(* PLC project CHL-DZ-BJDX-11 宁波数字孪生（东方理工）研究院制备薄层色谱全自动化工作站_Old_InoProShop(V1.9.1.6).project, Inovance company InoProShop(V1.9.1.6) InoProShop(V1.9.1.6) *)
(* stored: creationDateTime 2026-06-16T17:55:18.1932567, modificationDateTime 2026-06-04T10:59:46 *)

VAR_GLOBAL  (* HMI_Date *)
  HMI_HandWheel_3Y : BOOL;  (* 手轮切换 *)
  HMI_HandWheel_4X : BOOL;
  HMI_HandWheel_5Z : BOOL;
  HMI_HandWheel_6X : BOOL;
  HMI_HandWheel_7Y : BOOL;
  HMI_HandWheel_8Y : BOOL;
  HMI_HandWheel_9X : BOOL;
  HMI_HandWheel_10Z : BOOL;
  HMI_HandWheel_11Y : BOOL;
  一键回原点 : BOOL;
  伺服上料_Setp : INT;
  伺服下料_Setp : INT;
  HMI_打样瓶上料轴3Y AT %MB132240 : HMI_Servo;  (* <GrpComment>\r\n <GrpComment_zh-cn><Sub/>{k:["[[1,10]]","position","write","execute"],s:{1:{t:"0",s:["1行","2行","3行","4行","5行","6行","上料位"]},2:{t:"0",s:["1行","2行","3行","4行","5行","6行","上料位"]},3:{t:"0",s:["1行","2行","3行","4行","5行","6行","上料位"]}}}</GrpComment_zh-cn>\r\n <GrpComment_1><Sub/></GrpComment_1>\r\n <GrpComment_2><Sub/></GrpComment_2>\r\n </GrpComment> *)
  HMI_点样轴6X AT %MB132344 : HMI_Servo;  (* <GrpComment>\r\n <GrpComment_zh-cn><Sub/>{k:["[[1,10]]","position","write","execute"],s:{1:{t:"0",s:["清洗位","起始位","终点位"]},2:{t:"0",s:["清洗位","起始位","终点位"]},3:{t:"0",s:["清洗位","起始位","终点位"]}}}</GrpComment_zh-cn>\r\n <GrpComment_1><Sub/></GrpComment_1>\r\n <GrpComment_2><Sub/></GrpComment_2>\r\n </GrpComment> *)
  HMI_点样轴7Y AT %MB132448 : HMI_Servo;  (* <GrpComment>\r\n <GrpComment_zh-cn><Sub/>{k:["[[1,10]]","position","write","execute"],s:{1:{t:"0",s:["放板位","起始位"]},2:{t:"0",s:["放板位","起始位"]},3:{t:"0",s:["放板位","起始位"]}}}</GrpComment_zh-cn>\r\n <GrpComment_1><Sub/></GrpComment_1>\r\n <GrpComment_2><Sub/></GrpComment_2>\r\n </GrpComment> *)
  HMI_地轨轴11Y AT %MB132552 : HMI_Servo;  (* <GrpComment>\r\n <GrpComment_zh-cn><Sub/>{k:["[[1,10]]","position","write","execute"],s:{1:{t:"0",s:["上样点样位","刮板拍照位","收集位","取工具位","展开位","取收集组位"]},2:{t:"0",s:["上样点样位","刮板拍照位","收集位","取工具位","展开位","取收集组位"]},3:{t:"0",s:["上样点样位","刮板拍照位","收集位","取工具位","展开位","取收集组位"]}}}\r\n </GrpComment_zh-cn>\r\n <GrpComment_1><Sub/></GrpComment_1>\r\n <GrpComment_2><Sub/></GrpComment_2>\r\n </GrpComment> *)
  HMI_上样轴4X轴 AT %MB132656 : HMI_Servo;  (* <GrpComment>\r\n <GrpComment_zh-cn><Sub/>{k:["[[1,10]]","position","write","execute"],s:{1:{t:"0",s:["1列","2列","3列","4列","5列","6列","7列","8列","清洗位"]},2:{t:"0",s:["1列","2列","3列","4列","5列","6列","7列","8列","清洗位"]},3:{t:"0",s:["1列","2列","3列","4列","5列","6列","7列","8列",\r\n "清洗位"]}}}</GrpComment_zh-cn>\r\n <GrpComment_1><Sub/></GrpComment_1>\r\n <GrpComment_2><Sub/></GrpComment_2>\r\n </GrpComment> *)
  HMI_上样轴5Z轴 AT %MB132760 : HMI_Servo;  (* <GrpComment>\r\n <GrpComment_zh-cn><Sub/>{k:["[[1,10]]","position","write","execute"],s:{1:{t:"0",s:["清洗位","上液位"]},2:{t:"0",s:["清洗位","上液位"]},3:{t:"0",s:["清洗位","上液位"]}}}</GrpComment_zh-cn>\r\n <GrpComment_1><Sub/></GrpComment_1>\r\n <GrpComment_2><Sub/></GrpComment_2>\r\n </GrpComment> *)
  收集流程 : INT;
  收集计数 : INT;
  展开流程 : INT;
  上样点样流程 : INT;
  拍照刮板流程 : INT;
  机器人流程 : INT;
  升降上料完成 AT %MB132040 : BOOL;
  升降下料完成 AT %MB132041 : BOOL;
  ECAT掉站报警 : BOOL;
END_VAR

VAR_GLOBAL  (* cyinder_date *)
  cyinderAlarm : INT;
  cyinderAlarm2 : INT;
  展缸1气缸1手动 : BOOL;
  展缸1气缸1自动 : BOOL;
  展缸1气缸2手动 : BOOL;
  展缸1气缸2自动 : BOOL;
  展缸1气缸3手动 : BOOL;
  展缸1气缸3自动 : BOOL;
  展缸1气缸4手动 : BOOL;
  展缸1气缸4自动 : BOOL;
  展缸2气缸1手动 : BOOL;
  展缸2气缸1自动 : BOOL;
  展缸2气缸2手动 : BOOL;
  展缸2气缸2自动 : BOOL;
  展缸2气缸3手动 : BOOL;
  展缸2气缸3自动 : BOOL;
  展缸2气缸4手动 : BOOL;
  展缸2气缸4自动 : BOOL;
  收集下压气缸手动 : BOOL;
  收集下压气缸自动 : BOOL;
  收集夹持气缸手动 : BOOL;
  收集夹持气缸自动 : BOOL;
  收集升降气缸手动 : BOOL;
  收集升降气缸自动 : BOOL;
  收集伸缩气缸手动 : BOOL;
  收集伸缩气缸自动 : BOOL;
  刮板拍照遮光气缸手动 : BOOL;
  刮板拍照遮光气缸自动 : BOOL;
  刮板拍照旋转气缸手动 : BOOL;
  刮板拍照旋转气缸自动 : BOOL;
  刮板拍照下压气缸手动 : BOOL;
  刮板拍照下压气缸自动 : BOOL;
  展缸1进液电池阀1手动 : BOOL;
  展缸1进液电池阀1自动 : BOOL;
  展缸1进液电池阀2手动 : BOOL;
  展缸1进液电池阀2自动 : BOOL;
  展缸1进液电池阀3手动 : BOOL;
  展缸1进液电池阀3自动 : BOOL;
  展缸1进液电池阀4手动 : BOOL;
  展缸1进液电池阀4自动 : BOOL;
  展缸1排液电池阀1手动 : BOOL;
  展缸1排液电池阀1自动 : BOOL;
  展缸1排液电池阀2手动 : BOOL;
  展缸1排液电池阀2自动 : BOOL;
  展缸1排液电池阀3手动 : BOOL;
  展缸1排液电池阀3自动 : BOOL;
  展缸1排液电池阀4手动 : BOOL;
  展缸1排液电池阀4自动 : BOOL;
  展缸1吹气电池阀1手动 : BOOL;
  展缸1吹气电池阀1自动 : BOOL;
  展缸1吹气电池阀2手动 : BOOL;
  展缸1吹气电池阀2自动 : BOOL;
  展缸1吹气电池阀3手动 : BOOL;
  展缸1吹气电池阀3自动 : BOOL;
  展缸1吹气电池阀4手动 : BOOL;
  展缸1吹气电池阀4自动 : BOOL;
  大真空泵手动 : BOOL;
  大真空泵自动 : BOOL;
  展缸2进液电池阀1手动 : BOOL;
  展缸2进液电池阀1自动 : BOOL;
  展缸2进液电池阀2手动 : BOOL;
  展缸2进液电池阀2自动 : BOOL;
  展缸2进液电池阀3手动 : BOOL;
  展缸2进液电池阀3自动 : BOOL;
  展缸2进液电池阀4手动 : BOOL;
  展缸2进液电池阀4自动 : BOOL;
  展缸2排液电池阀1手动 : BOOL;
  展缸2排液电池阀1自动 : BOOL;
  展缸2排液电池阀2手动 : BOOL;
  展缸2排液电池阀2自动 : BOOL;
  展缸2排液电池阀3手动 : BOOL;
  展缸2排液电池阀3自动 : BOOL;
  展缸2排液电池阀4手动 : BOOL;
  展缸2排液电池阀4自动 : BOOL;
  展缸2吹气电池阀1手动 : BOOL;
  展缸2吹气电池阀1自动 : BOOL;
  展缸2吹气电池阀2手动 : BOOL;
  展缸2吹气电池阀2自动 : BOOL;
  展缸2吹气电池阀3手动 : BOOL;
  展缸2吹气电池阀3自动 : BOOL;
  展缸2吹气电池阀4手动 : BOOL;
  展缸2吹气电池阀4自动 : BOOL;
  收集进液手动 : BOOL;
  收集进液自动 : BOOL;
  收集排液手动 : BOOL;
  收集排液自动 : BOOL;
  收集正压排液手动 : BOOL;
  收集正压排液自动 : BOOL;
  溶液收集瓶定位手动 : BOOL;
  溶液收集瓶定位自动 : BOOL;
  上样定位手动 : BOOL;
  上样定位自动 : BOOL;
  上样点样三通电池阀手动 : BOOL;
  上样点样三通电池阀自动 : BOOL;
  刮板拍照真空手动 : BOOL;
  刮板拍照真空自动 : BOOL;
  刮板拍照无刷电机手动 : BOOL;
  刮板拍照无刷电机自动 : BOOL;
  刮板拍照定位气缸手动 : BOOL;
  刮板拍照定位气缸自动 : BOOL;
  粉末收集器定位手动 : BOOL;
  粉末收集器定位自动 : BOOL;
  上样吹气手动 : BOOL;
  上样吹气自动 : BOOL;
END_VAR

VAR_GLOBAL  (* IO *)
  A相 AT %IX0.0 : BOOL;
  B相 AT %IX0.1 : BOOL;
  急停 AT %IX0.3 : BOOL;
  复位 AT %IX0.4 : BOOL;
  启动 AT %IX0.5 : BOOL;
  停止 AT %IX0.6 : BOOL;
  手自动 AT %IX0.7 : BOOL;
  倍率X1 AT %IX1.0 : BOOL;
  倍率X10 AT %IX1.1 : BOOL;
  倍率X100 AT %IX1.2 : BOOL;
  选择轴1 AT %IX1.3 : BOOL;
  选择轴2 AT %IX1.4 : BOOL;
  选择轴3 AT %IX1.5 : BOOL;
  选择轴4 AT %IX1.6 : BOOL;
  三色灯红 AT %QX0.0 : BOOL;
  三色灯黄 AT %QX0.1 : BOOL;
  三色灯绿 AT %QX0.2 : BOOL;
  蜂鸣器 AT %QX0.3 : BOOL;
  展缸1进液电池阀1 AT %QX1.0 : BOOL;
  展缸1进液电池阀2 AT %QX1.1 : BOOL;
  展缸1进液电池阀3 AT %QX1.2 : BOOL;
  展缸1进液电池阀4 AT %QX1.3 : BOOL;
  展缸1排液电池阀1 AT %QX1.4 : BOOL;
  展缸1排液电池阀2 AT %QX1.5 : BOOL;
  展缸1排液电池阀3 AT %QX1.6 : BOOL;
  展缸1排液电池阀4 AT %QX1.7 : BOOL;
  展缸1吹气电池阀1 AT %QX2.0 : BOOL;
  展缸1吹气电池阀2 AT %QX2.1 : BOOL;
  展缸1吹气电池阀3 AT %QX2.2 : BOOL;
  展缸1吹气电池阀4 AT %QX2.3 : BOOL;
  大真空泵 AT %QX2.4 : BOOL;
  展缸2进液电池阀1 AT %QX3.0 : BOOL;
  展缸2进液电池阀2 AT %QX3.1 : BOOL;
  展缸2进液电池阀3 AT %QX3.2 : BOOL;
  展缸2进液电池阀4 AT %QX3.3 : BOOL;
  展缸2排液电池阀1 AT %QX3.4 : BOOL;
  展缸2排液电池阀2 AT %QX3.5 : BOOL;
  展缸2排液电池阀3 AT %QX3.6 : BOOL;
  展缸2排液电池阀4 AT %QX3.7 : BOOL;
  展缸2吹气电池阀1 AT %QX4.0 : BOOL;
  展缸2吹气电池阀2 AT %QX4.1 : BOOL;
  展缸2吹气电池阀3 AT %QX4.2 : BOOL;
  展缸2吹气电池阀4 AT %QX4.3 : BOOL;
  收集平台进液2通电池阀 AT %QX5.0 : BOOL;
  收集平台排液3通电池阀 AT %QX5.1 : BOOL;
  收集平台正压排液阀 AT %QX5.2 : BOOL;
  溶液收集瓶工位定位气缸 AT %QX5.3 : BOOL;
  上样定位气缸 AT %QX7.0 : BOOL;
  上样点样三通电池阀 AT %QX7.1 : BOOL;
  刮板拍照真空阀 AT %QX7.2 : BOOL;
  刮板拍照无刷电机 AT %QX7.3 : BOOL;
  刮板拍照定位气缸 AT %QX7.4 : BOOL;
  粉末收集器工位定位气缸 AT %QX7.5 : BOOL;
  上样吹气二通阀 AT %QX7.6 : BOOL;
  展缸1气缸1原点 AT %IX3.0 : BOOL;
  展缸1气缸1动点 AT %IX3.1 : BOOL;
  展缸1气缸2原点 AT %IX3.2 : BOOL;
  展缸1气缸2动点 AT %IX3.3 : BOOL;
  展缸1气缸3原点 AT %IX3.4 : BOOL;
  展缸1气缸3动点 AT %IX3.5 : BOOL;
  展缸1气缸4原点 AT %IX3.6 : BOOL;
  展缸1气缸4动点 AT %IX3.7 : BOOL;
  展缸1排液气泡传感器 AT %IX4.0 : BOOL;
  展缸1溶剂废液检测传感器 AT %IX4.1 : BOOL;
  展缸2气缸1原点 AT %IX5.0 : BOOL;
  展缸2气缸1动点 AT %IX5.1 : BOOL;
  展缸2气缸2原点 AT %IX5.2 : BOOL;
  展缸2气缸2动点 AT %IX5.3 : BOOL;
  展缸2气缸3原点 AT %IX5.4 : BOOL;
  展缸2气缸3动点 AT %IX5.5 : BOOL;
  展缸2气缸4原点 AT %IX5.6 : BOOL;
  展缸2气缸4动点 AT %IX5.7 : BOOL;
  展缸2排液气泡传感器 AT %IX6.0 : BOOL;
  展缸2溶剂废液检测传感器 AT %IX6.1 : BOOL;
  收集平台下压气缸原点 AT %IX7.0 : BOOL;
  上料进料传感器 AT %IX7.1 : BOOL;
  收集平台夹持气缸原点 AT %IX7.2 : BOOL;
  收集平台夹持气缸动点 AT %IX7.3 : BOOL;
  收集平台升降气缸原点 AT %IX7.4 : BOOL;
  收集平台升降气缸动点 AT %IX7.5 : BOOL;
  收集平台推出气缸原点 AT %IX7.6 : BOOL;
  收集平台推出气缸动点 AT %IX7.7 : BOOL;
  收集平台气泡传感器 AT %IX8.0 : BOOL;
  收集平台瓶子有无传感器 AT %IX8.1 : BOOL;
  收集平台暂存工位传感器 AT %IX8.2 : BOOL;
  玻璃升降光电开关1 AT %IX8.3 : BOOL;
  玻璃升降光电开关2 AT %IX8.4 : BOOL;
  玻璃升降接近开关1 AT %IX8.5 : BOOL;
  玻璃升降接近开关2 AT %IX8.6 : BOOL;
  下料出料传感器 AT %IX8.7 : BOOL;
  上样料架检测1 AT %IX9.0 : BOOL;
  上样料架检测2 AT %IX9.1 : BOOL;
  上样气泡传感器 AT %IX9.2 : BOOL;
  点样气泡传感器 AT %IX9.3 : BOOL;
  刮板拍照遮光气缸上位 AT %IX9.4 : BOOL;
  刮板拍照遮光气缸下位 AT %IX9.5 : BOOL;
  刮板拍照旋转气缸原点 AT %IX9.6 : BOOL;
  刮板拍照旋转气缸动点 AT %IX9.7 : BOOL;
  刮板拍照下压气缸上位 AT %IX10.0 : BOOL;
  刮板拍照暂存工位传感器 AT %IX10.2 : BOOL;
  料库检测1 AT %IX11.0 : BOOL;
  料库检测2 AT %IX11.1 : BOOL;
  料库检测3 AT %IX11.2 : BOOL;
  料库检测4 AT %IX11.3 : BOOL;
  料库检测5 AT %IX11.4 : BOOL;
  料库检测6 AT %IX11.5 : BOOL;
  料库检测7 AT %IX11.6 : BOOL;
  料库检测8 AT %IX11.7 : BOOL;
  料库检测9 AT %IX12.0 : BOOL;
  料库检测10 AT %IX12.1 : BOOL;
  料库检测11 AT %IX12.2 : BOOL;
  料库检测12 AT %IX12.3 : BOOL;
  机器人工具检测1 AT %IX12.4 : BOOL;
  机器人工具检测2 AT %IX12.5 : BOOL;
  机器人工具检测3 AT %IX12.6 : BOOL;
END_VAR

VAR_GLOBAL RETAIN PERSISTENT  (* servoaxisdate *)
  玻璃上料轴1ZDATE AT %MB131072 : servo;
  玻璃上料轴2ZDATE AT %MB131160 : servo;
  打样瓶上料轴3YDATE AT %MB131248 : servo;
  点样轴6XDATE AT %MB131336 : servo;
  点样轴7YDATE AT %MB131424 : servo;
  拍照轴8YDATE AT %MB131512 : servo;
  刮板轴9XDATE AT %MB131600 : servo;
  刮板轴10ZDATE AT %MB131688 : servo;
  地轨轴11YDATE AT %MB131776 : servo;
  上样轴4X轴DATE AT %MB131864 : servo;
  上样轴5Z轴DATE AT %MB131952 : servo;
END_VAR

VAR_GLOBAL  (* GVL *)
  MODE_State : INT;
  Alarm : INT;  (* 0:停止 1:运行 2:故障 3:急停 *)
  ManualAuto : BOOL;
  初始化 : BOOL;
  转发转存 AT %MW1301 : STRING(128);
  接收字符 AT %MW1001 : STRING(128);
  CNC启动 : BOOL;
  CNC停止 : BOOL;
  CNC完成 : BOOL;
  伺服报警 : BOOL;
  回零完成1Z : BOOL;
  回零完成2Z : BOOL;
  回零完成3Y : BOOL;
  回零完成4X : BOOL;
  回零完成5Z : BOOL;
  回零完成6X : BOOL;
  回零完成7Y : BOOL;
  回零完成8Y : BOOL;
  回零完成9X : BOOL;
  回零完成10Z : BOOL;
  回零完成11Y : BOOL;
  伺服未回原点报警 : BOOL;
  collect_prepare_OK : BOOL;
  collect_OK : BOOL;
  Camera_scraper_initialization_OK : BOOL;
  Photo_preparation_completed_OK : BOOL;
  Scraper_collection_completed : BOOL;
  Robot_completes_material_retrieval : BOOL;
  Sampling_initialization_OK : BOOL;
  Sampling_Cleaning_OK : BOOL;
  Sampling_preparation_OK : BOOL;
  Sampling_Place_materials_OK : BOOL;
  Sampling_liquid_absorption : BOOL;
  Sampling_Spray_sample_OK : BOOL;
  expand_initialization_OK : BOOL;
  Expand_Group_clean_OK : BOOL;
  Expand_up_liquid_OK : BOOL;
  Expand_silica_gel_plate_OK : BOOL;
  排液开始 : BOOL;
  Collector_coordinates : INT;
  Collect_bottle_coordinates : INT;
  上样清洗位置 : INT;
  取工具setp : INT;
  取工具完成 : BOOL;
  取升降硅胶板step : INT;
  取升降硅胶板完成 : BOOL;
  放点样硅胶板step : INT;
  放点样硅胶板完成 : BOOL;
  取点样硅胶板step : INT;
  取点样硅胶板完成 : BOOL;
  放展缸硅胶板完成 : BOOL;
  放展缸硅胶板step : INT;
  取展缸硅胶板step : INT;
  取展缸硅胶板完成 : BOOL;
  放拍照硅胶板完成 : BOOL;
  放拍照硅胶板step : INT;
  取收集器组放暂存工位step : INT;
  取收集瓶组放暂存工位完成 : BOOL;
  取暂存收集器放刮板位完成 : BOOL;
  取暂存收集器放刮板位step : INT;
  取刮板收集器放到收集工位完成 : BOOL;
  取刮板收集器放到收集工位step : INT;
  取暂存收集瓶放收集工位step : INT;
  取暂存收集瓶放收集工位完成 : BOOL;
  取收集器放暂存工位完成 : BOOL;
  取收集器放暂存工位step : INT;
  取刮板硅胶板放废料区step : INT;
  取刮板硅胶板放废料区完成 : BOOL;
  取暂存收集器组放仓库完成 : BOOL;
  取暂存收集器组放仓库step : INT;
  取收集器组放暂存工位完成 : BOOL;
  取收集瓶组放暂存工位step : INT;
  取暂存收集瓶组放仓库完成 : BOOL;
  取暂存收集瓶组放仓库step : INT;
  取收集瓶放暂存工位step : INT;
  取收集瓶放暂存工位完成 : BOOL;
  B1 : ARRAY[1..2000] OF SMC_GEOINFO;
  泵站位符 : BOOL;
  B2 : ARRAY[1..2000] OF SMC_GEOINFO;
  DR : INT;
  大真空泵站位 : ARRAY[0..11] OF BOOL;
  取拍照硅胶完step : INT;
  取拍照硅胶板完成 : BOOL;
  上样料架报警 : BOOL;
  bParameterList1 : ARRAY[1..8] OF BOOL;
  Z1JOG_pos : BOOL;
  Z1JOG_neg : BOOL;
  Z2JOG_POS : BOOL;
  Z2JOG_NEG : BOOL;
END_VAR

VAR_GLOBAL  (* Host_Computer *)
  bOutput : BOOL;
  bEnable : BOOL := TRUE;
  bErrorReset : BOOL;
  bStepEnable : BOOL := TRUE;
  PLC_Busy : BOOL := FALSE;  (* <GrpComment>\r\n <GrpComment_zh-cn>PLC 正在执行动作</GrpComment_zh-cn>\r\n </GrpComment>\r\n PLC 正在执行动作 *)
  collect_Done : BOOL := FALSE;  (* <GrpComment>\r\n <GrpComment_zh-cn>修改:动作执行完成</GrpComment_zh-cn>\r\n </GrpComment>\r\n 修改:动作执行完成 *)
  collect_Error : BOOL := FALSE;  (* <GrpComment>\r\n <GrpComment_zh-cn>新增：动作执行错误/急停</GrpComment_zh-cn>\r\n </GrpComment>\r\n 新增：动作执行错误/急停 *)
  PLC_EStop : BOOL;  (* <GrpComment>\r\n <GrpComment_zh-cn>新增：急停</GrpComment_zh-cn>\r\n </GrpComment>\r\n 新增：急停 *)
  collect_Reset : BOOL;  (* <GrpComment>\r\n <GrpComment_zh-cn>新增：收集工位置位</GrpComment_zh-cn>\r\n </GrpComment>\r\n 新增：收集工位置位 *)
  collect_Step : INT;  (* <GrpComment>\r\n <GrpComment_zh-cn>修改：收集工位状态机</GrpComment_zh-cn>\r\n </GrpComment>\r\n 修改：收集工位状态机 *)
  collect_forward_instructions : STRING(128);  (* <GrpComment>\r\n <GrpComment_zh-cn>收集工位注射泵转发指令</GrpComment_zh-cn>\r\n </GrpComment>\r\n 收集工位注射泵转发指令 *)
  collect_count : INT;  (* <GrpComment>\r\n <GrpComment_zh-cn>收集次数</GrpComment_zh-cn>\r\n </GrpComment>\r\n 收集次数 *)
  collect_Enable : BOOL;  (* <GrpComment>\r\n <GrpComment_zh-cn>新增：收集工位启动</GrpComment_zh-cn>\r\n </GrpComment>\r\n 新增：收集工位启动 *)
  collect_Busy : BOOL;  (* <GrpComment>\r\n <GrpComment_zh-cn>新增：收集工位忙</GrpComment_zh-cn>\r\n </GrpComment>\r\n 新增：收集工位忙 *)
  Expand_Enable : BOOL;  (* <GrpComment>\r\n <GrpComment_zh-cn>PC→PLC: TRUE 启动状态机</GrpComment_zh-cn>\r\n </GrpComment>\r\n PC→PLC: TRUE 启动状态机 *)
  Expand_Step : INT;  (* <GrpComment>\r\n <GrpComment_zh-cn>PLC→PC: 子步号 {0,10,20,30,40,90}</GrpComment_zh-cn>\r\n </GrpComment>\r\n PLC→PC: 子步号 {0,10,20,30,40,90} *)
  Expand_Done : BOOL;  (* <GrpComment>\r\n <GrpComment_zh-cn>PLC→PC: prep完成锁存（语义变更：prep完成非整流程完成）</GrpComment_zh-cn>\r\n </GrpComment>\r\n PLC→PC: prep完成锁存（语义变更：prep完成非整流程完成） *)
  Expand_Error : BOOL;  (* <GrpComment>\r\n <GrpComment_zh-cn>PLC→PC: 故障锁存（Step=90），Expand_Reset=TRUE 清零</GrpComment_zh-cn>\r\n </GrpComment>\r\n PLC→PC: 故障锁存（Step=90），Expand_Reset=TRUE 清零 *)
  Expand_Reset : BOOL;  (* <GrpComment>\r\n <GrpComment_zh-cn>PC→PLC: TRUE 清错误</GrpComment_zh-cn>\r\n </GrpComment>\r\n PC→PLC: TRUE 清错误 *)
  Expand_Busy : BOOL;  (* <GrpComment>\r\n <GrpComment_zh-cn>PLC→PC: 派生 (Step∈[10,80]) AND NOT Done</GrpComment_zh-cn>\r\n </GrpComment>\r\n PLC→PC: 派生 (Step∈[10,80]) AND NOT Done *)
  Expand_Mode_Flag : INT;  (* <GrpComment>\r\n <GrpComment_zh-cn>0=缸模式润洗 / 1=管路模式润洗</GrpComment_zh-cn>\r\n </GrpComment>\r\n 0=缸模式润洗 / 1=管路模式润洗 *)
  Expand_Group : INT;  (* <GrpComment>\r\n <GrpComment_zh-cn>展开组号 (1 或 2)，由 PLC 自动推导</GrpComment_zh-cn>\r\n </GrpComment>\r\n 展开组号 (1 或 2)，由 PLC 自动推导 *)
  Expand_Number : INT;  (* <GrpComment>\r\n <GrpComment_zh-cn>缸号在组内序号（1-4），由 PLC 自动推导</GrpComment_zh-cn>\r\n </GrpComment>\r\n 缸号在组内序号（1-4），由 PLC 自动推导 *)
  Expand_up_liquid_count : INT;  (* <GrpComment>\r\n <GrpComment_zh-cn>注射泵 DT 协议指令（合并后的单一变量）</GrpComment_zh-cn>\r\n </GrpComment>\r\n 上液注射泵重复次数 *)
  Expand_rinse_count : INT;  (* <GrpComment>\r\n <GrpComment_zh-cn>注射泵 DT 协议指令（合并后的单一变量）</GrpComment_zh-cn>\r\n </GrpComment>\r\n 润洗重复次数 *)
  Expand_forward_instructions : STRING(128);  (* <GrpComment>\r\n <GrpComment_zh-cn>注射泵 DT 协议指令（合并后的单一变量）</GrpComment_zh-cn>\r\n </GrpComment>\r\n 注射泵 DT 协议指令（合并后的单一变量） *)
  Tank_State : ARRAY[1..8] OF INT;  (* <GrpComment>\r\n <GrpComment_zh-cn>══════════════════════════════════════════════════════════════\r\n 【新增】展缸状态跟踪\r\n ══════════════════════════════════════════════════════════════</GrpComment_zh-cn>\r\n </GrpComment>\r\n ══════════════════════════════════════════════════════════════\r\n 【新增】展缸状态跟踪\r\n ══════════════════════════════════════════════════════════════ *)
  Tank_SampleID : ARRAY[1..8] OF DINT;  (* <GrpComment>\r\n <GrpComment_zh-cn>PLC→PC: 每缸状态\r\n 0 = Idle（空闲，可分配）\r\n 10 = Prepping（准备中：润洗/上液/放板）\r\n 40 = Developing（展开中，等待视觉/延时触发排液）\r\n 50 = Draining（排液中）\r\n 99 = Done（排液完成，等待 PC 释放）\r\n 90 = Error（故障）</GrpComment_zh-cn>\r\n </GrpComment>\r\n PLC→PC: 每缸状态\r\n 0 = Idle（空闲，可分配）\r\n 10 = Prepping（准备中：润洗/上液/放板）\r\n 40 = Developing（展开中，等待视觉/延时触发排液）\r\n 50 = Draining（排液中）\r\n 99 = Done（排液完成，等待 PC 释放）\r\n 90 = Error（故障） *)
  Expand_Target_Tank : INT;  (* <GrpComment>\r\n <GrpComment_zh-cn>PC→PLC: 绑定样品 ID（调试/溯源用，PLC 不使用此值做逻辑判断）\r\n ══════════════════════════════════════════════════════════════\r\n 【新增】Prep 目标参数\r\n ══════════════════════════════════════════════════════════════</GrpComment_zh-cn>\r\n </GrpComment>\r\n PC→PLC: 绑定样品 ID（调试/溯源用，PLC 不使用此值做逻辑判断）\r\n ══════════════════════════════════════════════════════════════\r\n 【新增】Prep 目标参数\r\n ══════════════════════════════════════════════════════════════ *)
  Tank_Drain_Enable : ARRAY[1..8] OF BOOL;  (* <GrpComment>\r\n <GrpComment_zh-cn>PC→PLC: 目标缸号(1-8)，Enable 触发前写入\r\n PLC 读取后自动推导：\r\n Expand_Group = (Target_Tank - 1) / 4 + 1\r\n Expand_Number = (Target_Tank - 1) MOD 4 + 1\r\n ══════════════════════════════════════════════════════════════\r\n 【新增】Per-tank 排液控制\r\n ══════════════════════════════════════════════════════════════</GrpComment_zh-cn>\r\n </GrpComment>\r\n PC→PLC: 目标缸号(1-8)，Enable 触发前写入\r\n PLC 读取后自动推导：\r\n Expand_Group = (Target_Tank - 1) / 4 + 1\r\n Expand_Number = (Target_Tank - 1) MOD 4 + 1\r\n ══════════════════════════════════════════════════════════════\r\n 【新增】Per-tank 排液控制\r\n ══════════════════════════════════════════════════════════════ *)
  Tank_Drain_Done : ARRAY[1..8] OF BOOL;  (* <GrpComment>\r\n <GrpComment_zh-cn>PC→PLC: 触发第 i 缸排液（前置条件：Tank_State[i]=40）</GrpComment_zh-cn>\r\n </GrpComment>\r\n PC→PLC: 触发第 i 缸排液（前置条件：Tank_State[i]=40） *)
  DrainTimer : ARRAY[1..8] OF TON;  (* <GrpComment>\r\n <GrpComment_zh-cn>PLC→PC: 第 i 缸排液完成锁存\r\n PC 确认后写 Tank_Drain_Enable[i]=FALSE 进行复位\r\n ══════════════════════════════════════════════════════════════\r\n 【新增】排液子程序内部变量\r\n ══════════════════════════════════════════════════════════════</GrpComment_zh-cn>\r\n </GrpComment>\r\n PLC→PC: 第 i 缸排液完成锁存\r\n PC 确认后写 Tank_Drain_Enable[i]=FALSE 进行复位\r\n ══════════════════════════════════════════════════════════════\r\n 【新增】排液子程序内部变量\r\n ══════════════════════════════════════════════════════════════ *)
  DrainDuration : TIME := TIME#5s0ms;  (* <GrpComment>\r\n <GrpComment_zh-cn>每缸排液定时器（后续可替换为传感器判断）</GrpComment_zh-cn>\r\n </GrpComment>\r\n 每缸排液定时器（后续可替换为传感器判断） *)
  Sampling_Enable : BOOL;  (* <GrpComment>\r\n <GrpComment_zh-cn>PC→PLC: TRUE 启动状态机</GrpComment_zh-cn>\r\n </GrpComment>\r\n PC→PLC: TRUE 启动状态机 *)
  Sampling_Step : INT;  (* <GrpComment>\r\n <GrpComment_zh-cn>PLC→PC: 子步号 {0,10,20,30,40,50,90}</GrpComment_zh-cn>\r\n </GrpComment>\r\n PLC→PC: 子步号 {0,10,20,30,40,50,90} *)
  Sampling_Done : BOOL;  (* <GrpComment>\r\n <GrpComment_zh-cn>PLC→PC: 完成锁存（Step 50 结束后置 TRUE）</GrpComment_zh-cn>\r\n </GrpComment>\r\n PLC→PC: 完成锁存（Step 50 结束后置 TRUE） *)
  Sampling_Error : BOOL;  (* <GrpComment>\r\n <GrpComment_zh-cn>PLC→PC: 故障锁存（Step=90），Sampling_Reset=TRUE 清零</GrpComment_zh-cn>\r\n </GrpComment>\r\n PLC→PC: 故障锁存（Step=90），Sampling_Reset=TRUE 清零 *)
  Sampling_Reset : BOOL;  (* <GrpComment>\r\n <GrpComment_zh-cn>PC→PLC: TRUE 清错误</GrpComment_zh-cn>\r\n </GrpComment>\r\n PC→PLC: TRUE 清错误 *)
  Sampling_Busy : BOOL;  (* <GrpComment>\r\n <GrpComment_zh-cn>PLC→PC: 派生 (Step∈[10,80]) AND NOT Done</GrpComment_zh-cn>\r\n </GrpComment>\r\n PLC→PC: 派生 (Step∈[10,80]) AND NOT Done *)
  Sampling_clean_instructions : ARRAY[1..2] OF STRING(128);  (* <GrpComment>\r\n <GrpComment_zh-cn>PC→PLC: 清洗泵指令（1条DT协议）</GrpComment_zh-cn>\r\n </GrpComment>\r\n PC→PLC: 清洗泵指令（1条DT协议） *)
  Sampling_clean_count : INT;  (* <GrpComment>\r\n <GrpComment_zh-cn>PC→PLC: 清洗次数（0=跳过清洗）</GrpComment_zh-cn>\r\n </GrpComment>\r\n PC→PLC: 清洗次数（0=跳过清洗） *)
  Sampling_prep_instructions : ARRAY[1..2] OF STRING(128);  (* <GrpComment>\r\n <GrpComment_zh-cn>── Step 20 气泡准备 ──</GrpComment_zh-cn>\r\n </GrpComment>\r\n 上样准备泵指令 *)
  Sampling_bubble_count : INT;  (* <GrpComment>\r\n <GrpComment_zh-cn>PC→PLC: 气泡序列指令数组，按 bubble_count 逐条执行\r\n 上位机 translate_sample_bubble_cmd() 生成，默认 Phase1=6条，上限 16</GrpComment_zh-cn>\r\n </GrpComment>\r\n PC→PLC: 气泡序列指令数组，按 bubble_count 逐条执行\r\n 上位机 translate_sample_bubble_cmd() 生成，默认 Phase1=6条，上限 16 *)
  Sampling_BubbleSensor : BOOL;  (* <GrpComment>\r\n <GrpComment_zh-cn>PC→PLC: 数组有效条目数（0=跳过气泡准备）</GrpComment_zh-cn>\r\n </GrpComment>\r\n PC→PLC: 数组有效条目数（0=跳过气泡准备） *)
  Sampling_phase2_instructions : STRING(128);  (* <GrpComment>\r\n <GrpComment_zh-cn>PLC 物理输入 / OPC UA 可写（调试用）\r\n TRUE = 气泡传感器检测到气-液界面到达上样针位置\r\n TODO【实机集成点】映射为物理输入 AT %IXx.y</GrpComment_zh-cn>\r\n </GrpComment>\r\n PLC 物理输入 / OPC UA 可写（调试用）\r\n TRUE = 气泡传感器检测到气-液界面到达上样针位置\r\n TODO【实机集成点】映射为物理输入 AT %IXx.y *)
  Sampling_Phase2_MaxCycles : INT;  (* <GrpComment>\r\n <GrpComment_zh-cn>PC→PLC: Phase 2 单次补液泵指令（循环执行直到传感器触发）\r\n 简化版未使用，实机需按 [pending]plc_spotting.txt Step 20 Phase 2 实现</GrpComment_zh-cn>\r\n </GrpComment>\r\n PC→PLC: Phase 2 单次补液泵指令（循环执行直到传感器触发）\r\n 简化版未使用，实机需按 [pending]plc_spotting.txt Step 20 Phase 2 实现 *)
  Sampling_X_coordinate : INT;  (* <GrpComment>\r\n <GrpComment_zh-cn>PC→PLC: 上样 X 坐标（逻辑索引，PLC内部查表映射物理坐标）</GrpComment_zh-cn>\r\n </GrpComment>\r\n PC→PLC: 上样 X 坐标（逻辑索引，PLC内部查表映射物理坐标） *)
  Sampling_Y_coordinate : INT;  (* <GrpComment>\r\n <GrpComment_zh-cn>PC→PLC: 上样 Y 坐标</GrpComment_zh-cn>\r\n </GrpComment>\r\n PC→PLC: 上样 Y 坐标 *)
  Sampling_sample_instructions : ARRAY[1..2] OF STRING(128);  (* <GrpComment>\r\n <GrpComment_zh-cn>PC→PLC: 吸液泵指令（1条DT协议）</GrpComment_zh-cn>\r\n </GrpComment>\r\n PC→PLC: 上样泵指令 *)
  Sampling_dispense_instructions : ARRAY[1..2] OF STRING(128);  (* <GrpComment>\r\n <GrpComment_zh-cn>PC→PLC: 点样泵指令（1条DT协议）</GrpComment_zh-cn>\r\n </GrpComment>\r\n PC→PLC: 点样泵指令（1条DT协议） *)
  scrape_Enable : BOOL;  (* <GrpComment>\r\n <GrpComment_zh-cn>PC→PLC: TRUE 启动状态机；FALSE 清 Done 回 idle</GrpComment_zh-cn>\r\n </GrpComment>\r\n PC→PLC: TRUE 启动状态机；FALSE 清 Done 回 idle *)
  scrape_Step : INT;  (* <GrpComment>\r\n <GrpComment_zh-cn>PLC→PC: 子步号 {0,10,15,20,30,40,90}</GrpComment_zh-cn>\r\n </GrpComment>\r\n PLC→PC: 子步号 {0,10,15,20,30,40,90} *)
  scrape_Done : BOOL;  (* <GrpComment>\r\n <GrpComment_zh-cn>PLC→PC: 完成锁存（Step 40 结束后置 TRUE）</GrpComment_zh-cn>\r\n </GrpComment>\r\n PLC→PC: 完成锁存（Step 40 结束后置 TRUE） *)
  scrape_Error : BOOL;  (* <GrpComment>\r\n <GrpComment_zh-cn>PLC→PC: 故障锁存（Step=90），scrape_Reset=TRUE 清零</GrpComment_zh-cn>\r\n </GrpComment>\r\n PLC→PC: 故障锁存（Step=90），scrape_Reset=TRUE 清零 *)
  scrape_Reset : BOOL;  (* <GrpComment>\r\n <GrpComment_zh-cn>PC→PLC: TRUE 清错误</GrpComment_zh-cn>\r\n </GrpComment>\r\n PC→PLC: TRUE 清错误 *)
  scrape_Busy : BOOL;  (* <GrpComment>\r\n <GrpComment_zh-cn>PLC→PC: 派生 (Step∈[10,80]) AND NOT Done</GrpComment_zh-cn>\r\n </GrpComment>\r\n PLC→PC: 派生 (Step∈[10,80]) AND NOT Done *)
  scrape_Confirm : BOOL;  (* <GrpComment>\r\n <GrpComment_zh-cn>PC→PLC: 乒乓确认信号</GrpComment_zh-cn>\r\n </GrpComment>\r\n PC→PLC: 乒乓确认信号 *)
  scrape_gcode_instructions : STRING(128);  (* <GrpComment>\r\n <GrpComment_zh-cn>PC→PLC: G-code 刮取路径指令</GrpComment_zh-cn>\r\n </GrpComment>\r\n PC→PLC: G-code 刮取路径指令 *)
  scrape_PhotoMode : INT;  (* <GrpComment>\r\n <GrpComment_zh-cn>PC→PLC: 拍照模式选择</GrpComment_zh-cn>\r\n </GrpComment>\r\n PC→PLC: 拍照模式选择 *)
  g_sx : ARRAY[1..400] OF REAL;
  g_sy : ARRAY[1..400] OF REAL;
  g_cx : ARRAY[1..400] OF REAL;
  g_cy : ARRAY[1..400] OF REAL;
  g_scrape_feed : INT;
  g_pass_count : INT;  (* 刮取次数 *)
  g_pass_z : REAL;  (* Z高度 *)
  IX0 AT %IB0 : BYTE;
  IX1 AT %IB1 : BYTE;
  IX2 AT %IB2 : BYTE;
  IX3 AT %IB3 : BYTE;
  IX4 AT %IB4 : BYTE;
  IX5 AT %IB5 : BYTE;
  IX6 AT %IB6 : BYTE;
  IX7 AT %IB7 : BYTE;
  IX8 AT %IB8 : BYTE;
  IX9 AT %IB9 : BYTE;
  IX10 AT %IB10 : BYTE;
  IX11 AT %IB11 : BYTE;
  IX12 AT %IB12 : BYTE;
  scrape_WaitConfirm : BOOL;  (* 允许拍照信号 *)
  collect_Fetch_Rack_Plate : INT;  (* 收集器取库位号 *)
  scrape_Fetch_Rack_Plate : INT;  (* 收集瓶料库号 *)
  collect_Consume_Slot : INT;  (* 取收集器料位号 *)
  collect_Powder_Return_Slot : INT;  (* 放收集器料位号 *)
  scrape_Consume_Slot : INT;  (* 收集瓶取放料位号 *)
  collect_Old_Plate_Slot : INT;  (* 收集器放库位号 *)
  scrape_Old_Plate_Slot : INT;  (* 收集瓶放库位号 *)
END_VAR

VAR_GLOBAL  (* RB_Date *)
  Execute : INT;  (* 0:FALSE 1:REUE *)
  Reset : INT;  (* 0:FALSE 1:REUE *)
  FunctionID : INT;  (* 0-255 *)
  ParameterList1 : INT;  (* 展开数据 *)
  ParameterList2 : INT;
  ParameterList3 : INT;
  ParameterList4 : INT;
  ParameterList5 : INT;
  ParameterList6 : INT;
  ParameterList7 : INT;
  ParameterList8 : INT;
  ParameterList9 : INT;  (* 0:Free 1:Busy 2:Complete 255:Error *)
  ParameterList10 : INT;  (* 0:Free 1:Busy 2:Complete 255:Error *)
  Status : INT;  (* 0:Free 1:Busy 2:Complete 255:Error *)
  Point : INT;  (* 0:原点初始化 1-255 自定义 *)
  ErrorID : INT;  (* <GrpComment>\r\n <GrpComment_zh-cn>0:无错误 255:不允许运行</GrpComment_zh-cn>\r\n </GrpComment>\r\n 0:无错误 255:不允许运行 *)
  RO_ParameterList1 : INT;
  RO_ParameterList2 : INT;
  RO_ParameterList3 : INT;
  RO_ParameterList4 : INT;
  RO_ParameterList5 : INT;
  RO_ParameterList6 : INT;
  RO_ParameterList7 : INT;
  RO_ParameterList8 : INT;
  RO_ParameterList9 : INT;
  RO_ParameterList10 : INT;
  收集工位允许放收集瓶 : BOOL;
  收集工位允许放收集器 : BOOL;
  收集工位放收集瓶完成 : BOOL;
  收集工位放收集器到工位 : BOOL;
  收集工位允许机器人退出工位 : BOOL;
  收集工位机器人退出完成 : BOOL;
  收集工位允许机器人取收集瓶放暂存工位 : BOOL;
  收集工位机器人放收集瓶到暂存工位完成 : BOOL;
  收集工位允许取收集器 : BOOL;
  收集工位机器人到达收集器位置 : BOOL;
  收集工位机器人取收集器放回暂存工位 : BOOL;
  收集工位放收集器完成 : BOOL;
  展开工位允许放硅胶板 : BOOL;
  展开工位允许取硅胶板 : BOOL;
  展开工位机器人到达准备点 : BOOL;
  展开工位机器人放硅胶板完成 : BOOL;
  展开工位取硅胶板完成 : BOOL;
  上样点样允许放硅胶板 : BOOL;
  上样点样允许取硅胶板 : BOOL;
  上样点样放硅胶板完成 : BOOL;
  拍照工位允许放硅胶板 : BOOL;
  拍照工位放硅胶板完成 : BOOL;
  拍照工位允许放收集器 : BOOL;
  拍照工位机器人到达夹持位 : BOOL;
  拍照工位机器人退出工位 : BOOL;
  拍照工位机器人退出工位完成 : BOOL;
  拍照工位允许取收集器 : BOOL;
  拍照工位机器人到达收集器夹持位 : BOOL;
  拍照工位机器人退出 : BOOL;
  拍照工位机器人退出完成 : BOOL;
  拍照工位允许取硅胶板放废料区 : BOOL;
  拍照工位允许取硅胶板去展开 : BOOL;
  拍照工位机器人取硅胶板完成 : BOOL;
  升降上料伺服允许取料 : BOOL;
  升降上料机器人已吸住物料 : BOOL;
  升降上料伺服下降完成 : BOOL;
  升降上料机器人取料完成 : BOOL;
  升降上料机器人放料完成 : BOOL;
  升降下料伺服允许放料 : BOOL;
  升降下料机器人放废料完成 : BOOL;
END_VAR
